(* IEC 61131-3 sources: 2026_Projet_YGO_ExcavatriceDragage/TOOLS/TWINBENCH/native_udp_poc, 4 files *)

(* ---- PRG_TwinBenchNativeUdp.st ---- *)
(* =======================================================================
   PRG_TwinBenchNativeUdp — POC transport UDP natif Control Win
   ───────────────────────────────────────────────────────────────
   🎯 Rôle : Mesurer un echo UDP loopback dans une tâche 10 ms isolée
   🔒 Polarité : Enable=FALSE ferme le socket ; aucun lien M3 ni sortie PLC
   🔌 Interface : SysSocket System, 127.0.0.1:29031/29032 uniquement
   ======================================================================= *)
PROGRAM PRG_TwinBenchNativeUdp
VAR
    // === COMMANDE POC ===
    Enable              : BOOL := FALSE;  // TRUE = mesure UDP locale active
    Stop                : BOOL := FALSE;  // TRUE = fermeture explicite socket

    // === ETAT PUBLIC ===
    SocketReady         : BOOL := FALSE;
    SentCount           : UDINT := 0;
    ReceivedCount       : UDINT := 0;
    SendErrorCount      : UDINT := 0;
    InvalidReplyCount   : UDINT := 0;
    LastResult          : SysTypes.RTS_IEC_RESULT := 0;
    LastBytesSent       : __XINT := 0;
    LastBytesReceived   : __XINT := 0;

    // === SOCKET PRIVE ===
    SocketHandle        : SysTypes.RTS_IEC_HANDLE := SysTypes.RTS_INVALID_HANDLE;
    NonBlocking         : DINT := 1;
    Reply               : UDP_REPLY;
    Tx                  : ARRAY [0..15] OF BYTE;
    Rx                  : ARRAY [0..15] OF BYTE;
    TxSequence          : UINT := 0;
END_VAR

// Le POC est inerte par défaut et ferme explicitement le port sous Control Win.
IF Stop OR NOT Enable THEN
    IF SocketHandle <> SysTypes.RTS_INVALID_HANDLE THEN
        SysSockCloseUdp(SocketHandle);
    END_IF;
    SocketHandle := SysTypes.RTS_INVALID_HANDLE;
    SocketReady := FALSE;
    RETURN;
END_IF;

// Un socket par programme, ports constants : destination 29031, retour 29032.
IF SocketHandle = SysTypes.RTS_INVALID_HANDLE THEN
    SocketHandle := SysSockCreateUdp(29031, 29032, ADR(LastResult));
    IF SocketHandle <> SysTypes.RTS_INVALID_HANDLE THEN
        LastResult := SysSockIoctl(SocketHandle, SOCKET_FIONBIO, ADR(NonBlocking));
        SocketReady := (LastResult = 0);
    END_IF;
    RETURN;
END_IF;

// Paquet fixe : "TB08", sequence UINT little-endian, reste reserve a zero.
Tx[0] := 16#54;
Tx[1] := 16#42;
Tx[2] := 16#30;
Tx[3] := 16#38;
Tx[4] := UINT_TO_BYTE(TxSequence AND 16#00FF);
Tx[5] := UINT_TO_BYTE(SHR(TxSequence, 8) AND 16#00FF);
Tx[6] := 0; Tx[7] := 0; Tx[8] := 0; Tx[9] := 0;
Tx[10] := 0; Tx[11] := 0; Tx[12] := 0; Tx[13] := 0;
Tx[14] := 0; Tx[15] := 0;

LastBytesSent := SysSockSendToUdp(SocketHandle, 29031, '127.0.0.1', ADR(Tx), SIZEOF(Tx), ADR(LastResult));
IF LastBytesSent = SIZEOF(Tx) THEN
    SentCount := SentCount + 1;
    TxSequence := TxSequence + 1;
ELSE
    SendErrorCount := SendErrorCount + 1;
END_IF;

// Non-bloquant : l'absence de réponse est normale au scan courant.
LastBytesReceived := SysSockRecvFromUdp(SocketHandle, ADR(Rx), SIZEOF(Rx), ADR(Reply), ADR(LastResult));
IF LastBytesReceived > 0 THEN
    IF (LastBytesReceived = SIZEOF(Rx))
       AND (Rx[0] = 16#54) AND (Rx[1] = 16#42)
       AND (Rx[2] = 16#30) AND (Rx[3] = 16#38) THEN
        ReceivedCount := ReceivedCount + 1;
    ELSE
        InvalidReplyCount := InvalidReplyCount + 1;
    END_IF;
END_IF;

(* ---- PRG_TwinBenchNativeUdpMulti.st ---- *)
(* =======================================================================
   PRG_TwinBenchNativeUdpMulti — POC UDP multi-flux Control Win
   ───────────────────────────────────────────────────────────────
   🎯 Rôle : Mesurer flux rapide/cyclique/événementiel sans bloquer la tâche
   🔒 Polarité : Enable=FALSE ou Stop=TRUE ferme les trois sockets
   🔌 Interface : SysSocket System, 127.0.0.1 uniquement, aucun lien machine
   ======================================================================= *)
PROGRAM PRG_TwinBenchNativeUdpMulti
VAR
    // === COMMANDE POC ===
    Enable              : BOOL := FALSE;
    Stop                : BOOL := FALSE;
    EventTrigger        : BOOL := FALSE;

    // === ETAT PUBLIC ===
    SocketReady         : BOOL := FALSE;
    FastSentCount       : UDINT := 0;
    FastReceivedCount   : UDINT := 0;
    CyclicSentCount     : UDINT := 0;
    CyclicReceivedCount : UDINT := 0;
    EventSentCount      : UDINT := 0;
    EventReceivedCount  : UDINT := 0;
    SendErrorCount      : UDINT := 0;
    InvalidReplyCount   : UDINT := 0;
    LastResult          : SysTypes.RTS_IEC_RESULT := 0;

    // === SOCKETS PRIVES ===
    FastSocket          : SysTypes.RTS_IEC_HANDLE := SysTypes.RTS_INVALID_HANDLE;
    CyclicSocket        : SysTypes.RTS_IEC_HANDLE := SysTypes.RTS_INVALID_HANDLE;
    EventSocket         : SysTypes.RTS_IEC_HANDLE := SysTypes.RTS_INVALID_HANDLE;
    NonBlocking         : DINT := 1;
    FastReply           : UDP_REPLY;
    CyclicReply         : UDP_REPLY;
    EventReply          : UDP_REPLY;
    FastTx              : ARRAY [0..15] OF BYTE;
    FastRx              : ARRAY [0..15] OF BYTE;
    CyclicTx            : ARRAY [0..15] OF BYTE;
    CyclicRx            : ARRAY [0..15] OF BYTE;
    EventTx             : ARRAY [0..15] OF BYTE;
    EventRx             : ARRAY [0..15] OF BYTE;
    FastSequence        : UINT := 0;
    CyclicSequence      : UINT := 0;
    EventSequence       : UINT := 0;
    CycleDivider        : USINT := 0;
    EventPrevious       : BOOL := FALSE;
    Bytes               : __XINT := 0;
END_VAR

IF Stop OR NOT Enable THEN
    IF FastSocket <> SysTypes.RTS_INVALID_HANDLE THEN SysSockCloseUdp(FastSocket); END_IF;
    IF CyclicSocket <> SysTypes.RTS_INVALID_HANDLE THEN SysSockCloseUdp(CyclicSocket); END_IF;
    IF EventSocket <> SysTypes.RTS_INVALID_HANDLE THEN SysSockCloseUdp(EventSocket); END_IF;
    FastSocket := SysTypes.RTS_INVALID_HANDLE;
    CyclicSocket := SysTypes.RTS_INVALID_HANDLE;
    EventSocket := SysTypes.RTS_INVALID_HANDLE;
    SocketReady := FALSE;
    EventPrevious := EventTrigger;
    RETURN;
END_IF;

// Initialisation progressive : le scan ne poursuit qu une fois les trois sockets prets.
IF FastSocket = SysTypes.RTS_INVALID_HANDLE THEN
    FastSocket := SysSockCreateUdp(29031, 29032, ADR(LastResult));
    IF FastSocket <> SysTypes.RTS_INVALID_HANDLE THEN LastResult := SysSockIoctl(FastSocket, SOCKET_FIONBIO, ADR(NonBlocking)); END_IF;
    RETURN;
END_IF;
IF CyclicSocket = SysTypes.RTS_INVALID_HANDLE THEN
    CyclicSocket := SysSockCreateUdp(29041, 29042, ADR(LastResult));
    IF CyclicSocket <> SysTypes.RTS_INVALID_HANDLE THEN LastResult := SysSockIoctl(CyclicSocket, SOCKET_FIONBIO, ADR(NonBlocking)); END_IF;
    RETURN;
END_IF;
IF EventSocket = SysTypes.RTS_INVALID_HANDLE THEN
    EventSocket := SysSockCreateUdp(29051, 29052, ADR(LastResult));
    IF EventSocket <> SysTypes.RTS_INVALID_HANDLE THEN LastResult := SysSockIoctl(EventSocket, SOCKET_FIONBIO, ADR(NonBlocking)); END_IF;
    SocketReady := (LastResult = 0);
    RETURN;
END_IF;

// Entete commun TB08, classe de flux en octet 6, sequence UINT en octets 4/5.
FastTx[0] := 16#54; FastTx[1] := 16#42; FastTx[2] := 16#30; FastTx[3] := 16#38;
FastTx[4] := UINT_TO_BYTE(FastSequence AND 16#00FF); FastTx[5] := UINT_TO_BYTE(SHR(FastSequence, 8) AND 16#00FF); FastTx[6] := 1;
Bytes := SysSockSendToUdp(FastSocket, 29031, '127.0.0.1', ADR(FastTx), SIZEOF(FastTx), ADR(LastResult));
IF Bytes = SIZEOF(FastTx) THEN FastSentCount := FastSentCount + 1; FastSequence := FastSequence + 1; ELSE SendErrorCount := SendErrorCount + 1; END_IF;

// Receptions toutes non bloquantes, meme quand leur emission est moins frequente.
Bytes := SysSockRecvFromUdp(FastSocket, ADR(FastRx), SIZEOF(FastRx), ADR(FastReply), ADR(LastResult));
IF Bytes > 0 THEN
    IF (Bytes = SIZEOF(FastRx)) AND (FastRx[0] = 16#54) AND (FastRx[6] = 1) THEN FastReceivedCount := FastReceivedCount + 1; ELSE InvalidReplyCount := InvalidReplyCount + 1; END_IF;
END_IF;

CycleDivider := CycleDivider + 1;
IF CycleDivider >= 5 THEN
    CycleDivider := 0;
    CyclicTx[0] := 16#54; CyclicTx[1] := 16#42; CyclicTx[2] := 16#30; CyclicTx[3] := 16#38;
    CyclicTx[4] := UINT_TO_BYTE(CyclicSequence AND 16#00FF); CyclicTx[5] := UINT_TO_BYTE(SHR(CyclicSequence, 8) AND 16#00FF); CyclicTx[6] := 2;
    Bytes := SysSockSendToUdp(CyclicSocket, 29041, '127.0.0.1', ADR(CyclicTx), SIZEOF(CyclicTx), ADR(LastResult));
    IF Bytes = SIZEOF(CyclicTx) THEN CyclicSentCount := CyclicSentCount + 1; CyclicSequence := CyclicSequence + 1; ELSE SendErrorCount := SendErrorCount + 1; END_IF;
END_IF;
Bytes := SysSockRecvFromUdp(CyclicSocket, ADR(CyclicRx), SIZEOF(CyclicRx), ADR(CyclicReply), ADR(LastResult));
IF Bytes > 0 THEN
    IF (Bytes = SIZEOF(CyclicRx)) AND (CyclicRx[0] = 16#54) AND (CyclicRx[6] = 2) THEN CyclicReceivedCount := CyclicReceivedCount + 1; ELSE InvalidReplyCount := InvalidReplyCount + 1; END_IF;
END_IF;

IF EventTrigger AND NOT EventPrevious THEN
    EventTx[0] := 16#54; EventTx[1] := 16#42; EventTx[2] := 16#30; EventTx[3] := 16#38;
    EventTx[4] := UINT_TO_BYTE(EventSequence AND 16#00FF); EventTx[5] := UINT_TO_BYTE(SHR(EventSequence, 8) AND 16#00FF); EventTx[6] := 3;
    Bytes := SysSockSendToUdp(EventSocket, 29051, '127.0.0.1', ADR(EventTx), SIZEOF(EventTx), ADR(LastResult));
    IF Bytes = SIZEOF(EventTx) THEN EventSentCount := EventSentCount + 1; EventSequence := EventSequence + 1; ELSE SendErrorCount := SendErrorCount + 1; END_IF;
END_IF;
EventPrevious := EventTrigger;
Bytes := SysSockRecvFromUdp(EventSocket, ADR(EventRx), SIZEOF(EventRx), ADR(EventReply), ADR(LastResult));
IF Bytes > 0 THEN
    IF (Bytes = SIZEOF(EventRx)) AND (EventRx[0] = 16#54) AND (EventRx[6] = 3) THEN EventReceivedCount := EventReceivedCount + 1; ELSE InvalidReplyCount := InvalidReplyCount + 1; END_IF;
END_IF;

(* ---- PRG_TwinBenchNativeUdpMulti_DECLARATION.st ---- *)
VAR
    // === COMMANDE POC ===
    Enable              : BOOL := FALSE;
    Stop                : BOOL := FALSE;
    EventTrigger        : BOOL := FALSE;

    // === ETAT PUBLIC ===
    SocketReady         : BOOL := FALSE;
    FastSentCount       : UDINT := 0;
    FastReceivedCount   : UDINT := 0;
    CyclicSentCount     : UDINT := 0;
    CyclicReceivedCount : UDINT := 0;
    EventSentCount      : UDINT := 0;
    EventReceivedCount  : UDINT := 0;
    SendErrorCount      : UDINT := 0;
    InvalidReplyCount   : UDINT := 0;
    LastResult          : SysTypes.RTS_IEC_RESULT := 0;

    // === SOCKETS PRIVES ===
    FastSocket          : SysTypes.RTS_IEC_HANDLE := SysTypes.RTS_INVALID_HANDLE;
    CyclicSocket        : SysTypes.RTS_IEC_HANDLE := SysTypes.RTS_INVALID_HANDLE;
    EventSocket         : SysTypes.RTS_IEC_HANDLE := SysTypes.RTS_INVALID_HANDLE;
    NonBlocking         : DINT := 1;
    FastReply           : UDP_REPLY;
    CyclicReply         : UDP_REPLY;
    EventReply          : UDP_REPLY;
    FastTx              : ARRAY [0..15] OF BYTE;
    FastRx              : ARRAY [0..15] OF BYTE;
    CyclicTx            : ARRAY [0..15] OF BYTE;
    CyclicRx            : ARRAY [0..15] OF BYTE;
    EventTx             : ARRAY [0..15] OF BYTE;
    EventRx             : ARRAY [0..15] OF BYTE;
    FastSequence        : UINT := 0;
    CyclicSequence      : UINT := 0;
    EventSequence       : UINT := 0;
    CycleDivider        : USINT := 0;
    EventPrevious       : BOOL := FALSE;
    Bytes               : __XINT := 0;
END_VAR

(* ---- PRG_TwinBenchNativeUdpMulti_IMPLEMENTATION.st ---- *)
IF Stop OR NOT Enable THEN
    IF FastSocket <> SysTypes.RTS_INVALID_HANDLE THEN SysSockCloseUdp(FastSocket); END_IF;
    IF CyclicSocket <> SysTypes.RTS_INVALID_HANDLE THEN SysSockCloseUdp(CyclicSocket); END_IF;
    IF EventSocket <> SysTypes.RTS_INVALID_HANDLE THEN SysSockCloseUdp(EventSocket); END_IF;
    FastSocket := SysTypes.RTS_INVALID_HANDLE;
    CyclicSocket := SysTypes.RTS_INVALID_HANDLE;
    EventSocket := SysTypes.RTS_INVALID_HANDLE;
    SocketReady := FALSE;
    EventPrevious := EventTrigger;
    RETURN;
END_IF;

IF FastSocket = SysTypes.RTS_INVALID_HANDLE THEN
    FastSocket := SysSockCreateUdp(29031, 29032, ADR(LastResult));
    IF FastSocket <> SysTypes.RTS_INVALID_HANDLE THEN LastResult := SysSockIoctl(FastSocket, SOCKET_FIONBIO, ADR(NonBlocking)); END_IF;
    RETURN;
END_IF;
IF CyclicSocket = SysTypes.RTS_INVALID_HANDLE THEN
    CyclicSocket := SysSockCreateUdp(29041, 29042, ADR(LastResult));
    IF CyclicSocket <> SysTypes.RTS_INVALID_HANDLE THEN LastResult := SysSockIoctl(CyclicSocket, SOCKET_FIONBIO, ADR(NonBlocking)); END_IF;
    RETURN;
END_IF;
IF EventSocket = SysTypes.RTS_INVALID_HANDLE THEN
    EventSocket := SysSockCreateUdp(29051, 29052, ADR(LastResult));
    IF EventSocket <> SysTypes.RTS_INVALID_HANDLE THEN LastResult := SysSockIoctl(EventSocket, SOCKET_FIONBIO, ADR(NonBlocking)); END_IF;
    SocketReady := (LastResult = 0);
    RETURN;
END_IF;

FastTx[0] := 16#54; FastTx[1] := 16#42; FastTx[2] := 16#30; FastTx[3] := 16#38;
FastTx[4] := UINT_TO_BYTE(FastSequence AND 16#00FF); FastTx[5] := UINT_TO_BYTE(SHR(FastSequence, 8) AND 16#00FF); FastTx[6] := 1;
Bytes := SysSockSendToUdp(FastSocket, 29031, '127.0.0.1', ADR(FastTx), SIZEOF(FastTx), ADR(LastResult));
IF Bytes = SIZEOF(FastTx) THEN FastSentCount := FastSentCount + 1; FastSequence := FastSequence + 1; ELSE SendErrorCount := SendErrorCount + 1; END_IF;

Bytes := SysSockRecvFromUdp(FastSocket, ADR(FastRx), SIZEOF(FastRx), ADR(FastReply), ADR(LastResult));
IF Bytes > 0 THEN
    IF (Bytes = SIZEOF(FastRx)) AND (FastRx[0] = 16#54) AND (FastRx[6] = 1) THEN FastReceivedCount := FastReceivedCount + 1; ELSE InvalidReplyCount := InvalidReplyCount + 1; END_IF;
END_IF;

CycleDivider := CycleDivider + 1;
IF CycleDivider >= 5 THEN
    CycleDivider := 0;
    CyclicTx[0] := 16#54; CyclicTx[1] := 16#42; CyclicTx[2] := 16#30; CyclicTx[3] := 16#38;
    CyclicTx[4] := UINT_TO_BYTE(CyclicSequence AND 16#00FF); CyclicTx[5] := UINT_TO_BYTE(SHR(CyclicSequence, 8) AND 16#00FF); CyclicTx[6] := 2;
    Bytes := SysSockSendToUdp(CyclicSocket, 29041, '127.0.0.1', ADR(CyclicTx), SIZEOF(CyclicTx), ADR(LastResult));
    IF Bytes = SIZEOF(CyclicTx) THEN CyclicSentCount := CyclicSentCount + 1; CyclicSequence := CyclicSequence + 1; ELSE SendErrorCount := SendErrorCount + 1; END_IF;
END_IF;
Bytes := SysSockRecvFromUdp(CyclicSocket, ADR(CyclicRx), SIZEOF(CyclicRx), ADR(CyclicReply), ADR(LastResult));
IF Bytes > 0 THEN
    IF (Bytes = SIZEOF(CyclicRx)) AND (CyclicRx[0] = 16#54) AND (CyclicRx[6] = 2) THEN CyclicReceivedCount := CyclicReceivedCount + 1; ELSE InvalidReplyCount := InvalidReplyCount + 1; END_IF;
END_IF;

IF EventTrigger AND NOT EventPrevious THEN
    EventTx[0] := 16#54; EventTx[1] := 16#42; EventTx[2] := 16#30; EventTx[3] := 16#38;
    EventTx[4] := UINT_TO_BYTE(EventSequence AND 16#00FF); EventTx[5] := UINT_TO_BYTE(SHR(EventSequence, 8) AND 16#00FF); EventTx[6] := 3;
    Bytes := SysSockSendToUdp(EventSocket, 29051, '127.0.0.1', ADR(EventTx), SIZEOF(EventTx), ADR(LastResult));
    IF Bytes = SIZEOF(EventTx) THEN EventSentCount := EventSentCount + 1; EventSequence := EventSequence + 1; ELSE SendErrorCount := SendErrorCount + 1; END_IF;
END_IF;
EventPrevious := EventTrigger;
Bytes := SysSockRecvFromUdp(EventSocket, ADR(EventRx), SIZEOF(EventRx), ADR(EventReply), ADR(LastResult));
IF Bytes > 0 THEN
    IF (Bytes = SIZEOF(EventRx)) AND (EventRx[0] = 16#54) AND (EventRx[6] = 3) THEN EventReceivedCount := EventReceivedCount + 1; ELSE InvalidReplyCount := InvalidReplyCount + 1; END_IF;
END_IF;
